// TIA Portal V20 export
// export: Created 2025-12-01T14:56:13.5765522Z, ExportSetting None, DisplayName Totally Integrated Automation Portal, DisplayVersion V20 Update 3, DisplayName TIA Portal Openness, DisplayVersion V20 Update 3, DisplayName TIA Portal Version Control Interface, DisplayVersion V20 Update 3, DisplayName STEP 7 Professional, DisplayVersion V20 Update 3, DisplayName STEP 7 Safety, DisplayVersion V20 Update 2, DisplayName WinCC Basic/Comfort/Advanced, DisplayVersion V20 Update 3, DisplayName WinCC Professional, DisplayVersion V20 Update 3, DisplayName WinCC Unified, DisplayVersion V20 Update 3
TYPE "UDT_EventosPantalla"
   STRUCT
      Mckey : UDInt;
      NivelVisual : UInt;
      LineaTexto_01 : String[48];   // Primer Linea del Texto a Visulizar
      LineaTexto_02 : String[48];   // Segunda Linea del Texto a Visulizar
      LineaTexto_03 : String[48];   // Tercera Linea del Texto a Visulizar
      LineaTexto_04 : String[48];   // Cuarta Linea del Texto a Visulizar
   END_STRUCT;
END_TYPE
